// TIA Portal V18 export
FUNCTION_BLOCK "Scenario1ReadWrite"   // FB5, FBD
{ S7_Optimized_Access := 'TRUE' }
AUTHOR : SIOS
FAMILY : LIOLink_AwB
// stored: IsIECCheckEnabled true, MemoryReserve 100, SetENOAutomatically true
   VAR_INPUT
      hwID : HW_IO;
      port123 : Int;
      readWrite : Bool;
      reqParameterPage0 : Bool;
      reqSystemCommands : Bool;
      reqVendorName : Bool;
      reqVendorText : Bool;
      reqProductName : Bool;
      reqProductID : Bool;
      reqSerialNumber : Bool;
      reqHwRevision : Bool;
      reqFwRevision : Bool;
      reqAppSpecificName : Bool;
      reqDiagnostics : Bool;
      reqMeasurements : Bool;
      reqParameters : Bool;
   END_VAR
   VAR_OUTPUT
      done { ExternalWritable := 'False'} : Bool;
      busy { ExternalWritable := 'False'} : Bool;
      error { ExternalWritable := 'False'} : Bool;
      status { ExternalWritable := 'False'} : Word;
      diagDeviceFb { ExternalWritable := 'False'} : "LIOLink_typeDiagnostics";
   END_VAR
   VAR_IN_OUT
      data : "LIOLink_3RR24_typeAll";
   END_VAR
   VAR
      statReq { ExternalAccessible := 'False'; ExternalVisible := 'False'; ExternalWritable := 'False'} : Bool;
      instCurrMonitorRelay { ExternalAccessible := 'False'; ExternalVisible := 'False'; ExternalWritable := 'False'} : "LIOLink_3RR24";
   END_VAR
BEGIN

REGION Network 1
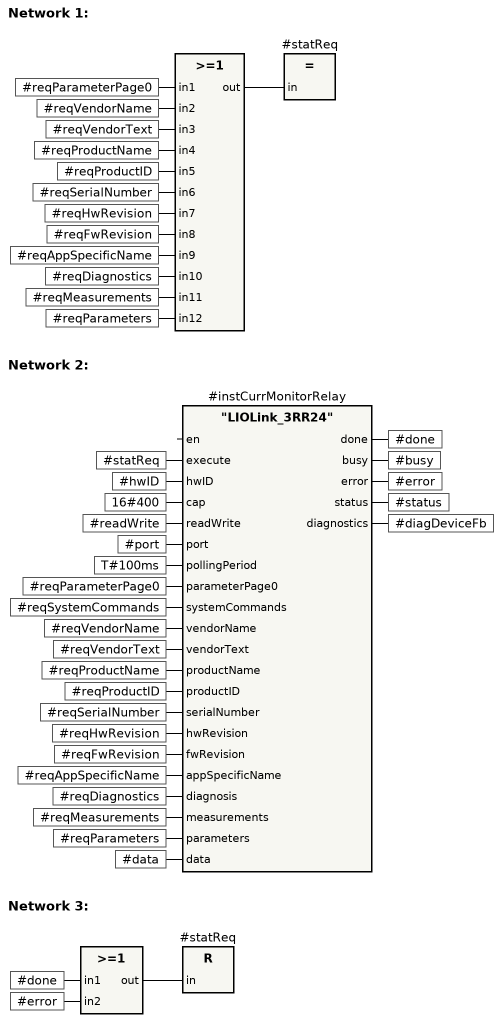
   #statReq := #reqParameterPage0 OR #reqVendorName OR #reqVendorText OR #reqProductName OR #reqProductID OR #reqSerialNumber OR #reqHwRevision OR #reqFwRevision OR #reqAppSpecificName OR #reqDiagnostics OR #reqMeasurements OR #reqParameters;
END_REGION

REGION Network 2
   #instCurrMonitorRelay(execute := #statReq,   // "LIOLink_3RR24"
                         hwID := #hwID,
                         cap := 16#400,
                         readWrite := #readWrite,
                         port := #port,
                         pollingPeriod := T#100ms,
                         parameterPage0 := #reqParameterPage0,
                         systemCommands := #reqSystemCommands,
                         vendorName := #reqVendorName,
                         vendorText := #reqVendorText,
                         productName := #reqProductName,
                         productID := #reqProductID,
                         serialNumber := #reqSerialNumber,
                         hwRevision := #reqHwRevision,
                         fwRevision := #reqFwRevision,
                         appSpecificName := #reqAppSpecificName,
                         diagnosis := #reqDiagnostics,
                         measurements := #reqMeasurements,
                         parameters := #reqParameters,
                         data := #data,
                         done => #done,
                         busy => #busy,
                         error => #error,
                         status => #status,
                         diagnostics => #diagDeviceFb);
END_REGION

REGION Network 3
   IF #done OR #error THEN #statReq := FALSE; END_IF;
END_REGION
END_FUNCTION_BLOCK
